PROGRAM MAIN
VAR
END_VAR

END_PROGRAM

(* stored: Version 1.1.0.1, ProductVersion 3.1.4024.12
   POU MAIN: Id {28dc04ef-af3b-4cf4-870f-3cdbdb932f7c}, SpecialFunc None *)
